{attribute 'linkalways'} 
{attribute 'no_explicit_call' := 'This FB is a CLASS and must be accessed using methods or properties'}
{attribute 'enable_dynamic_creation'}
FUNCTION_BLOCK FINAL LE_DWORD EXTENDS Node
VAR
	in1 : _DWORD(0);
	in2 : _DWORD(0);
	out : _BOOL(FALSE);
END_VAR

METHOD PUBLIC Clone : I_Node
VAR
	pNode : POINTER TO LE_DWORD;
END_VAR
pNode := __NEW(LE_DWORD);
Clone := pNode^;
END_METHOD

METHOD FB_init : BOOL
VAR_INPUT
	bInitRetains : BOOL; // if TRUE, the retain variables are initialized (warm start / cold start)
	bInCopyCode : BOOL;  // if TRUE, the instance afterwards gets moved into the copy code (online change)
END_VAR
AddInput('in1',THIS^.in1);
AddInput('in2',THIS^.in2);
AddOutput('out', THIS^.out);
END_METHOD

METHOD PROTECTED OnExecute
VAR
END_VAR
out.Value := in1.Value <= in2.Value;
END_METHOD

END_FUNCTION_BLOCK

(* stored: Version 1.1.0.1, ProductVersion 3.1.4024.15
   POU LE_DWORD: Id {ad2fd77a-20c2-4b39-a241-20c397acdd8b}, SpecialFunc None
   Folder Constructor: Id {68e6d37c-6250-449d-8b4f-aa17ea365905}
   Method Clone: Id {cca75abb-a368-4711-8156-7dbc36241474}
   Method FB_init: Id {3879f069-8ada-4f16-b658-767547df3856}
   Method OnExecute: Id {3c7ada3c-1459-45ba-977c-9aa3e33441f2} *)
